// TIA Portal V20 export
TYPE "mz_LOGSOperationData1"
// stored: Access Published
   STRUCT
      ReadyForOperation : Bool;
      MachineInOperation : Bool;
      NoInterference : Bool;
      RequestPart : Bool;
      NoPart : Bool;
   END_STRUCT;
END_TYPE
